{attribute addProperty BoxType "EL6001--0000"}
{attribute addProperty Id "CtrlAT %Q*UINT1621Data_OutAT %Q*ARRAY[0 ..21] OF USINT176220"}
{attribute addProperty CRC "1274078981"}
{attribute addProperty SizeInBites "192"}
{attribute addProperty SizeInBytes "24"}
TYPE Outputs_377610EF :
STRUCT
	{attribute addProperty Name "Ctrl"}
	Ctrl AT %Q* : UINT;
	{attribute addProperty Name "Data_Out"}
	Data_Out AT %Q* : ARRAY[0 ..21] OF USINT;
END_STRUCT
END_TYPE

(* stored: Version 1.2.0.0, ProductVersion 3.1.4024.9
   DUT Outputs_377610EF: Id {cc4f25d1-aa63-4871-bc7f-8632d67af025} *)
